TYPE ST_DB_CACCheckCtrl :
STRUCT
	bDB_ExecuteCacCheck			: BOOL;
	bDB_CACCheckComplete		: BOOL;
	bDB_CaseOk					: BOOL;
	bDB_Error						: BOOL;
	stCacToCheck					: ST_CAC_Data;
END_STRUCT
END_TYPE

(* stored: Version 1.1.0.1
   DUT ST_DB_CACCheckCtrl: Id {f921fc95-419d-4d17-93be-ae6cd946c1b4} *)
